// TIA Portal V18 export
// export: Created 2025-12-01T12:38:05.6038445Z, ExportSetting None, DisplayName Totally Integrated Automation Portal, DisplayVersion V18 Update 5, DisplayName TIA Portal Openness, DisplayVersion V18 Update 5, DisplayName TIA Portal Teamcenter Gateway, DisplayVersion V18, DisplayName TIA Portal Version Control Interface, DisplayVersion V18, DisplayName STEP 7 Professional, DisplayVersion V18 Update 5, DisplayName STEP 7 Safety, DisplayVersion V18, DisplayName WinCC Professional, DisplayVersion V18 Update 5
DATA_BLOCK "ST10_TipDB"   // DB1069
{ S7_Optimized_Access := 'FALSE' }
// stored: AutoNumber false
   VAR RETAIN
      Global : Struct
         "1" : Struct
            ControlOn : Bool;   // 7000:提示：设备未上电，请先按复位按钮，再按控制开按钮
            closesafetyDoor : Bool;   // 7001:提示：设备存在故障，请查看报警信息，消除故障，然后按复位按钮
            LockSafetyDoor : Bool;   // 7003:提示：设备未选择自动，请选择自动模式
            SelectAutoMode : Bool;   // 7005:提示：设备未启动，请启动自动运行
            SelectManualMode : Bool;
            AutoModeRunning : Bool;
            SafetyDoorLocked : Bool;
            SaferyDoorNotLocked : Bool;
            GoWP : Bool;
            Reset : Bool;
         END_STRUCT;
         "2" : Array[0..15] of Bool;
         "3" : Array[0..15] of Bool;
         "4" : Array[0..15] of Bool;
         "5" : Struct
            FuncrionDeactive1 : Bool;
            FuncrionDeactive2 : Bool;
            FuncrionDeactive3 : Bool;
            FuncrionDeactive4 : Bool;
            FuncrionDeactive5 : Bool;
            FuncrionDeactive6 : Bool;
            FuncrionDeactive7 : Bool;
            FuncrionDeactive8 : Bool;
         END_STRUCT;
         "6" : Array[0..15] of Bool;
         "7" : Struct
            ScanMainPartDMC1 : Bool;
            ScanPartDMC2 : Bool;
            ScanPartDMC3 : Bool;
            ScanPartDMC4 : Bool;
            ScanPartDMC5 : Bool;
            ScanPartDMC6 : Bool;
            ScanPartDMC7 : Bool;
            ScanPartDMC8 : Bool;
         END_STRUCT;
         "8" : Array[0..15] of Bool;
         "9" : Array[0..15] of Bool;
         "10" : Array[0..15] of Bool;
      END_STRUCT;
      OP1 : Struct   // ST70_B_提示信息
         "Take off product" : Bool;   // 请取下托盘上产品
         "Put product" : Bool;   // 请放入转向器壳体总成
         "Please scan the code" : Bool;   // 请扫转向器壳体总成二维码
         "Please apply Oil" : Bool;   // 请手持涂油工装涂油
         "Please take the O-ring" : Bool;   // 请取O型圈并安装完成
         "Please put in the powertrain" : Bool;   // 请扫转向器总成二维码
         Static_2 : Bool;
         "Please pre-screw" : Bool;   // 请安装转向器动力总成并预拧螺丝
         Static_1 : Bool;
         Static_3 : Bool;
         "Please press the button_1" : Bool;   // 请按下ST70-B启动按钮
         Reset : Bool;   // RFID状态数据未清除，请复位清除数据
      END_STRUCT;
      OP2 : Struct   // ST70_C_提示信息
         Static_4 : Bool;
         Static_2 : Bool;
         Static_3 : Bool;
         "Please press the button" : Bool;   // 请按下ST70_C启动按钮
         "Please press the trigger" : Bool;   // 请按下螺丝枪扳机拧紧螺丝
         "Please take the paint pen" : Bool;   // 请取出油漆笔划上标识
         "Please put back the paint pen" : Bool;   // 请划上标识后放回油漆笔
         Static_1 : Bool;
         "Please remove the product" : Bool;   // 产品报废,请取下产品
         "Please press the screw gun trigger" : Bool;   // 重新拧紧,请按下螺丝枪扳机
      END_STRUCT;
   END_VAR
BEGIN
   // Global."2"[0] : 7002:提示：未选择配方，请在换型页面选择配方
   // Global."2"[1] : 7004:提示：设备未初始化，请启动初始化
END_DATA_BLOCK
